FUNCTION_BLOCK TcaRobotStorage EXTENDS TcaStorage 

VAR	
	nOriginId			: INT := -1;	
	eApproachDirection	: E_ApproachDirection;
	stSupportPoint		: ST_Coordinate;
	sPose				: STRING;
	
	bCarrierTeached		: ARRAY[0..nMaxCarrierTypes] OF BOOL;
	aOffset				: ARRAY[0..nMaxCarrierTypes] OF ST_Coordinate;
END_VAR

PROPERTY ApproachDirection : E_ApproachDirection
GET
ApproachDirection := eApproachDirection;
END_GET
SET
eApproachDirection := ApproachDirection;
END_SET
END_PROPERTY

PROPERTY OriginId : INT
GET
OriginId := nOriginId;
END_GET
SET
nOriginId := OriginId;
END_SET
END_PROPERTY

PROPERTY Pose : STRING
GET
Pose := sPose;
END_GET
SET
sPose := Pose;
END_SET
END_PROPERTY

METHOD RobotCoordinatesOf : ST_Coordinate
VAR_INPUT
	Position			: INT;
END_VAR

VAR
	tmpCoordinate		: ST_Coordinate;
END_VAR
IF NOT bCarrierPresent OR NOT bCarrierTeached[_Carrier.CarrierId] OR nOriginId = -1 THEN
	RETURN;
END_IF

tmpCoordinate := _Carrier.CoordinatesOf(Position);

tmpCoordinate.nOriginId := nOriginId;
tmpCoordinate.fX := tmpCoordinate.fX + aOffset[_Carrier.CarrierId].fX;
tmpCoordinate.fY := tmpCoordinate.fY + aOffset[_Carrier.CarrierId].fY;
tmpCoordinate.fZ := tmpCoordinate.fZ + aOffset[_Carrier.CarrierId].fZ;
tmpCoordinate.fRx := tmpCoordinate.fRx + aOffset[_Carrier.CarrierId].fRx;
tmpCoordinate.fRy := tmpCoordinate.fRy + aOffset[_Carrier.CarrierId].fRy;
tmpCoordinate.fRz := tmpCoordinate.fRz + aOffset[_Carrier.CarrierId].fRz;

RobotCoordinatesOf := tmpCoordinate;
END_METHOD

PROPERTY SupportPoint : ST_Coordinate
GET
SupportPoint := stSupportPoint;
END_GET
SET
stSupportPoint := SupportPoint;
END_SET
END_PROPERTY

METHOD TeachCarrierType : TcoCore.ITcoTaskStatus
VAR_INPUT
	CarrierId					: INT;	
	Offset_X					: REAL;	
	Offset_Y					: REAL;	
	Offset_Z					: REAL;	
	Offset_Rx					: REAL;	
	Offset_Ry					: REAL;	
	Offset_Rz					: REAL;
END_VAR
aOffset[CarrierId].fX := Offset_X;
aOffset[CarrierId].fY := Offset_Y;
aOffset[CarrierId].fZ := Offset_Z;
aOffset[CarrierId].fRx := Offset_Rx;
aOffset[CarrierId].fRy := Offset_Ry;
aOffset[CarrierId].fRz := Offset_Rz;

bCarrierTeached[CarrierId] := TRUE;
END_METHOD

END_FUNCTION_BLOCK

(* stored: Version 1.1.0.1
   POU TcaRobotStorage: Id {2e5f7d9e-e053-4b8b-959f-778fc713336b}, SpecialFunc None
   Property ApproachDirection: Id {5ba719f7-12b1-490c-a2e7-e0334c5e14a7}
   Get Get: Id {e0228633-da1d-423f-943c-372cd219180f}
   Set Set: Id {26c8c4ec-a593-4eb4-b866-61ab75173a24}
   Property OriginId: Id {8f864130-6e61-403d-9126-d270c762a499}
   Get Get: Id {b3ebb342-0f5e-4401-815d-b29fcf151682}
   Set Set: Id {828c749e-9b81-4192-bbb3-d17dd769c27c}
   Property Pose: Id {38bbae77-1584-4dec-b56c-47f23cbd5c2c}
   Get Get: Id {71146d90-8041-4d61-8055-42f5661f6a7e}
   Set Set: Id {5d27d215-6fc6-48c3-9028-ba4c391c9e8d}
   Method RobotCoordinatesOf: Id {83fd7b48-e261-44a3-9c9b-e078d9965116}
   Property SupportPoint: Id {33327287-8e5f-4bdb-9bdb-79bfae402714}
   Get Get: Id {73906dac-ae8c-4bd7-8b5f-e5c44279bd8c}
   Set Set: Id {3ed28bd4-d081-49b3-b581-94c81fa3bdf8}
   Method TeachCarrierType: Id {b3602fcb-dc42-43eb-9367-56c7ea30625b} *)
